# EPICS autosave request: andorApp/Db/shamrock_settings.req
$(P)$(R)SlitSize1
$(P)$(R)SlitSize2
$(P)$(R)SlitSize3
$(P)$(R)SlitSize4
$(P)$(R)FlipperMirror1
$(P)$(R)FlipperMirror2
